{attribute 'TcRpcEnable' := '1'}
METHOD start
  VAR_INPUT
    position : LREAL;  (* New position setpoint *)
    maxVelocity : LREAL;  (* Maximum velocity *)
  END_VAR
                  THIS^.get.position := position;
THIS^.get.maxVelocity := maxVelocity;
THIS^.statuses.busyStatus( isBusy := TRUE );
THIS^.statuses.healthStatus( isGood := TRUE );

                
END_METHOD

{attribute 'TcRpcEnable' := '1'}
METHOD request : RequestResults
  VAR_INPUT
    position : LREAL;  (* New position setpoint *)
    maxVelocity : LREAL;  (* Maximum velocity *)
  END_VAR
                  IF THIS^.statuses.enabledStatus.enabled THEN
    THIS^.start(
        position := position,
        maxVelocity := maxVelocity);
    request := RequestResults.ACCEPTED;
ELSE
    request := RequestResults.REJECTED;
END_IF;

                
END_METHOD
END_FUNCTION_BLOCK

FUNCTION_BLOCK McMoveRelativeProcess EXTENDS BaseMcProcess
  VAR_INPUT
    {attribute 'OPC.UA.DA' := '1'}
    set : McMoveRelativeProcessArgs;  (* Arguments to be set, before writing do_request TRUE *)
  END_VAR
  VAR_OUTPUT
    {attribute 'OPC.UA.DA' := '1'}
    {attribute 'OPC.UA.DA.Access' := '1'}
    get : McMoveRelativeProcessArgs;  (* Arguments in use by the process, if do_request was accepted *)
  END_VAR

            IF do_request THEN
    do_request_result := request(
    distance := set.distance,
    maxVelocity := set.maxVelocity);
    do_request := FALSE;
END_IF;
SUPER^();

          

{attribute 'TcRpcEnable' := '1'}
METHOD start
  VAR_INPUT
    distance : LREAL;  (* Distance to move *)
    maxVelocity : LREAL;  (* Maximum velocity *)
  END_VAR
                  THIS^.get.distance := distance;
THIS^.get.maxVelocity := maxVelocity;
THIS^.statuses.busyStatus( isBusy := TRUE );
THIS^.statuses.healthStatus( isGood := TRUE );

                
END_METHOD

{attribute 'TcRpcEnable' := '1'}
METHOD request : RequestResults
  VAR_INPUT
    distance : LREAL;  (* Distance to move *)
    maxVelocity : LREAL;  (* Maximum velocity *)
  END_VAR
                  IF THIS^.statuses.enabledStatus.enabled THEN
    THIS^.start(
        distance := distance,
        maxVelocity := maxVelocity);
    request := RequestResults.ACCEPTED;
ELSE
    request := RequestResults.REJECTED;
END_IF;

                
END_METHOD
END_FUNCTION_BLOCK

FUNCTION_BLOCK McPowerProcess EXTENDS BaseMcProcess
  VAR_INPUT
    {attribute 'OPC.UA.DA' := '1'}
    set : McPowerProcessArgs;  (* Arguments to be set, before writing do_request TRUE *)
  END_VAR
  VAR_OUTPUT
    {attribute 'OPC.UA.DA' := '1'}
    {attribute 'OPC.UA.DA.Access' := '1'}
    get : McPowerProcessArgs;  (* Arguments in use by the process, if do_request was accepted *)
  END_VAR

            IF do_request THEN
    do_request_result := request( enable := set.enable );
    do_request := FALSE;
END_IF;
SUPER^();

          

{attribute 'TcRpcEnable' := '1'}
METHOD start
  VAR_INPUT
    enable : BOOL;  (* Enable the power or not *)
  END_VAR
                  THIS^.get.enable := enable;
THIS^.statuses.busyStatus( isBusy := TRUE );
THIS^.statuses.healthStatus( isGood := TRUE );

                
END_METHOD

{attribute 'TcRpcEnable' := '1'}
METHOD request : RequestResults
  VAR_INPUT
    enable : BOOL;  (* Enable the power or not *)
  END_VAR
                  IF THIS^.statuses.enabledStatus.enabled THEN
    THIS^.start( enable := enable );
    request := RequestResults.ACCEPTED;
ELSE
    request := RequestResults.REJECTED;
END_IF;

                
END_METHOD
END_FUNCTION_BLOCK

FUNCTION_BLOCK McSetPositionProcess EXTENDS BaseMcProcess
  VAR_INPUT
    {attribute 'OPC.UA.DA' := '1'}
    set : McSetPositionProcessArgs;  (* Arguments to be set, before writing do_request TRUE *)
  END_VAR
  VAR_OUTPUT
    {attribute 'OPC.UA.DA' := '1'}
    {attribute 'OPC.UA.DA.Access' := '1'}
    get : McSetPositionProcessArgs;  (* Arguments in use by the process, if do_request was accepted *)
  END_VAR

            IF do_request THEN
    do_request_result := request( value := set.value );
    do_request := FALSE;
END_IF;
SUPER^();

          

{attribute 'TcRpcEnable' := '1'}
METHOD start
  VAR_INPUT
    value : LREAL;  (* New position to be taken over by the encoder *)
  END_VAR
                  THIS^.get.value := value;
THIS^.statuses.busyStatus( isBusy := TRUE );
THIS^.statuses.healthStatus( isGood := TRUE );

                
END_METHOD

{attribute 'TcRpcEnable' := '1'}
METHOD request : RequestResults
  VAR_INPUT
    value : LREAL;  (* New position to be taken over by the encoder *)
  END_VAR
                  IF THIS^.statuses.enabledStatus.enabled THEN
    THIS^.start( value := value );
    request := RequestResults.ACCEPTED;
ELSE
    request := RequestResults.REJECTED;
END_IF;

                
END_METHOD
END_FUNCTION_BLOCK

FUNCTION_BLOCK McStopProcess EXTENDS BaseMcProcess
  VAR_INPUT
    {attribute 'OPC.UA.DA' := '1'}
    set : McStopProcessArgs;  (* Arguments to be set, before writing do_request TRUE *)
  END_VAR
  VAR_OUTPUT
    {attribute 'OPC.UA.DA' := '1'}
    {attribute 'OPC.UA.DA.Access' := '1'}
    get : McStopProcessArgs;  (* Arguments in use by the process, if do_request was accepted *)
  END_VAR

            IF do_request THEN
    do_request_result := request(
    deceleration := set.deceleration,
    jerk := set.jerk);
    do_request := FALSE;
END_IF;
SUPER^();

          

{attribute 'TcRpcEnable' := '1'}
METHOD start
  VAR_INPUT
    deceleration : LREAL;  (* Deceleration (use 0 for default). If non zero, then also jerk must be non zero! *)
    jerk : LREAL;  (* Jerk (use 0 for default). If non zero, then also deceleration must be non zero! *)
  END_VAR
                  THIS^.get.deceleration := deceleration;
THIS^.get.jerk := jerk;
THIS^.statuses.busyStatus( isBusy := TRUE );
THIS^.statuses.healthStatus( isGood := TRUE );

                
END_METHOD

{attribute 'TcRpcEnable' := '1'}
METHOD request : RequestResults
  VAR_INPUT
    deceleration : LREAL;  (* Deceleration (use 0 for default). If non zero, then also jerk must be non zero! *)
    jerk : LREAL;  (* Jerk (use 0 for default). If non zero, then also deceleration must be non zero! *)
  END_VAR
                  IF THIS^.statuses.enabledStatus.enabled THEN
    THIS^.start(
        deceleration := deceleration,
        jerk := jerk);
    request := RequestResults.ACCEPTED;
ELSE
    request := RequestResults.REJECTED;
END_IF;

                
END_METHOD
END_FUNCTION_BLOCK

FUNCTION_BLOCK McMoveVelocityProcess EXTENDS BaseMcProcess
  VAR_INPUT
    {attribute 'OPC.UA.DA' := '1'}
    set : McMoveVelocityProcessArgs;  (* Arguments to be set, before writing do_request TRUE *)
  END_VAR
  VAR_OUTPUT
    {attribute 'OPC.UA.DA' := '1'}
    {attribute 'OPC.UA.DA.Access' := '1'}
    get : McMoveVelocityProcessArgs;  (* Arguments in use by the process, if do_request was accepted *)
  END_VAR

            IF do_request THEN
    do_request_result := request( value := set.value );
    do_request := FALSE;
END_IF;
SUPER^();

          

{attribute 'TcRpcEnable' := '1'}
METHOD start
  VAR_INPUT
    value : LREAL;  (* New velocity *)
  END_VAR
                  THIS^.get.value := value;
THIS^.statuses.busyStatus( isBusy := TRUE );
THIS^.statuses.healthStatus( isGood := TRUE );

                
END_METHOD

{attribute 'TcRpcEnable' := '1'}
METHOD request : RequestResults
  VAR_INPUT
    value : LREAL;  (* New velocity *)
  END_VAR
                  IF THIS^.statuses.enabledStatus.enabled THEN
    THIS^.start( value := value );
    request := RequestResults.ACCEPTED;
ELSE
    request := RequestResults.REJECTED;
END_IF;

                
END_METHOD
END_FUNCTION_BLOCK

FUNCTION_BLOCK SetEnabledProcess EXTENDS BaseProcess
  VAR_INPUT
    {attribute 'OPC.UA.DA' := '1'}
    set : SetEnabledProcessArgs;  (* Arguments to be set, before writing do_request TRUE *)
  END_VAR
  VAR_OUTPUT
    {attribute 'OPC.UA.DA' := '1'}
    {attribute 'OPC.UA.DA.Access' := '1'}
    get : SetEnabledProcessArgs;  (* Arguments in use by the process, if do_request was accepted *)
  END_VAR

            IF do_request THEN
    do_request_result := request( enabled := set.enabled );
    do_request := FALSE;
END_IF;
SUPER^();

          

{attribute 'TcRpcEnable' := '1'}
METHOD start
  VAR_INPUT
    enabled : BOOL;  (* True to enable, false to disable *)
  END_VAR
                  THIS^.get.enabled := enabled;
THIS^.statuses.busyStatus( isBusy := TRUE );
THIS^.statuses.healthStatus( isGood := TRUE );

                
END_METHOD

{attribute 'TcRpcEnable' := '1'}
METHOD request : RequestResults
  VAR_INPUT
    enabled : BOOL;  (* True to enable, false to disable *)
  END_VAR
                  IF THIS^.statuses.enabledStatus.enabled THEN
    THIS^.start( enabled := enabled );
    request := RequestResults.ACCEPTED;
ELSE
    request := RequestResults.REJECTED;
END_IF;

                
END_METHOD
END_FUNCTION_BLOCK

FUNCTION_BLOCK McWriteParameter EXTENDS BaseMcProcess
  VAR_INPUT
    {attribute 'OPC.UA.DA' := '1'}
    set : McWriteParameterArgs;  (* Arguments to be set, before writing do_request TRUE *)
  END_VAR
  VAR_OUTPUT
    {attribute 'OPC.UA.DA' := '1'}
    {attribute 'OPC.UA.DA.Access' := '1'}
    get : McWriteParameterArgs;  (* Arguments in use by the process, if do_request was accepted *)
  END_VAR

            IF do_request THEN
    do_request_result := request(
    parameterNumber := set.parameterNumber,
    value := set.value);
    do_request := FALSE;
END_IF;
SUPER^();

          

{attribute 'TcRpcEnable' := '1'}
METHOD start
  VAR_INPUT
    parameterNumber : INT;  (* Number of the parameter *)
    value : LREAL;  (* Value to write *)
  END_VAR
                  THIS^.get.parameterNumber := parameterNumber;
THIS^.get.value := value;
THIS^.statuses.busyStatus( isBusy := TRUE );
THIS^.statuses.healthStatus( isGood := TRUE );

                
END_METHOD

{attribute 'TcRpcEnable' := '1'}
METHOD request : RequestResults
  VAR_INPUT
    parameterNumber : INT;  (* Number of the parameter *)
    value : LREAL;  (* Value to write *)
  END_VAR
                  IF THIS^.statuses.enabledStatus.enabled THEN
    THIS^.start(
        parameterNumber := parameterNumber,
        value := value);
    request := RequestResults.ACCEPTED;
ELSE
    request := RequestResults.REJECTED;
END_IF;

                
END_METHOD
END_FUNCTION_BLOCK

FUNCTION_BLOCK McReadParameter EXTENDS BaseMcProcess
  VAR_INPUT
    value : LREAL;  (* Value that was read *)
    {attribute 'OPC.UA.DA' := '1'}
    set : McReadParameterArgs;  (* Arguments to be set, before writing do_request TRUE *)
  END_VAR
  VAR_OUTPUT
    {attribute 'OPC.UA.DA' := '1'}
    {attribute 'OPC.UA.DA.Access' := '1'}
    get : McReadParameterArgs;  (* Arguments in use by the process, if do_request was accepted *)
  END_VAR

            IF do_request THEN
    do_request_result := request( parameterNumber := set.parameterNumber );
    do_request := FALSE;
END_IF;
SUPER^();

          

{attribute 'TcRpcEnable' := '1'}
METHOD start
  VAR_INPUT
    parameterNumber : INT;  (* Number of the parameter *)
  END_VAR
                  THIS^.get.parameterNumber := parameterNumber;
THIS^.statuses.busyStatus( isBusy := TRUE );
THIS^.statuses.healthStatus( isGood := TRUE );

                
END_METHOD

{attribute 'TcRpcEnable' := '1'}
METHOD request : RequestResults
  VAR_INPUT
    parameterNumber : INT;  (* Number of the parameter *)
  END_VAR
                  IF THIS^.statuses.enabledStatus.enabled THEN
    THIS^.start( parameterNumber := parameterNumber );
    request := RequestResults.ACCEPTED;
ELSE
    request := RequestResults.REJECTED;
END_IF;

                
END_METHOD
END_FUNCTION_BLOCK

FUNCTION_BLOCK McWriteBoolParameter EXTENDS BaseMcProcess
  VAR_INPUT
    {attribute 'OPC.UA.DA' := '1'}
    set : McWriteBoolParameterArgs;  (* Arguments to be set, before writing do_request TRUE *)
  END_VAR
  VAR_OUTPUT
    {attribute 'OPC.UA.DA' := '1'}
    {attribute 'OPC.UA.DA.Access' := '1'}
    get : McWriteBoolParameterArgs;  (* Arguments in use by the process, if do_request was accepted *)
  END_VAR

            IF do_request THEN
    do_request_result := request(
    parameterNumber := set.parameterNumber,
    value := set.value);
    do_request := FALSE;
END_IF;
SUPER^();

          

{attribute 'TcRpcEnable' := '1'}
METHOD start
  VAR_INPUT
    parameterNumber : INT;  (* Number of the parameter *)
    value : BOOL;  (* Value to write *)
  END_VAR
                  THIS^.get.parameterNumber := parameterNumber;
THIS^.get.value := value;
THIS^.statuses.busyStatus( isBusy := TRUE );
THIS^.statuses.healthStatus( isGood := TRUE );

                
END_METHOD

{attribute 'TcRpcEnable' := '1'}
METHOD request : RequestResults
  VAR_INPUT
    parameterNumber : INT;  (* Number of the parameter *)
    value : BOOL;  (* Value to write *)
  END_VAR
                  IF THIS^.statuses.enabledStatus.enabled THEN
    THIS^.start(
        parameterNumber := parameterNumber,
        value := value);
    request := RequestResults.ACCEPTED;
ELSE
    request := RequestResults.REJECTED;
END_IF;

                
END_METHOD
END_FUNCTION_BLOCK

FUNCTION_BLOCK McReadBoolParameter EXTENDS BaseMcProcess
  VAR_INPUT
    value : BOOL;  (* Value that was read *)
    {attribute 'OPC.UA.DA' := '1'}
    set : McReadBoolParameterArgs;  (* Arguments to be set, before writing do_request TRUE *)
  END_VAR
  VAR_OUTPUT
    {attribute 'OPC.UA.DA' := '1'}
    {attribute 'OPC.UA.DA.Access' := '1'}
    get : McReadBoolParameterArgs;  (* Arguments in use by the process, if do_request was accepted *)
  END_VAR

            IF do_request THEN
    do_request_result := request( parameterNumber := set.parameterNumber );
    do_request := FALSE;
END_IF;
SUPER^();

          

{attribute 'TcRpcEnable' := '1'}
METHOD start
  VAR_INPUT
    parameterNumber : INT;  (* Number of the parameter *)
  END_VAR
                  THIS^.get.parameterNumber := parameterNumber;
THIS^.statuses.busyStatus( isBusy := TRUE );
THIS^.statuses.healthStatus( isGood := TRUE );

                
END_METHOD

{attribute 'TcRpcEnable' := '1'}
METHOD request : RequestResults
  VAR_INPUT
    parameterNumber : INT;  (* Number of the parameter *)
  END_VAR
                  IF THIS^.statuses.enabledStatus.enabled THEN
    THIS^.start( parameterNumber := parameterNumber );
    request := RequestResults.ACCEPTED;
ELSE
    request := RequestResults.REJECTED;
END_IF;

                
END_METHOD
END_FUNCTION_BLOCK

FUNCTION_BLOCK SDOReadProcess EXTENDS BaseProcess
  VAR_INPUT
    value1Byte : USINT;  (* Value that has been read, if noOfBytes is 1 *)
    value2Bytes : UINT;  (* Value that has been read, if noOfBytes is 2 *)
    value4Bytes : UDINT;  (* Value that has been read, if noOfBytes is 4 *)
    errorId : UDINT;  (* Error ID according to Beckhoff *)
    {attribute 'OPC.UA.DA' := '1'}
    set : SDOReadProcessArgs;  (* Arguments to be set, before writing do_request TRUE *)
  END_VAR
  VAR_OUTPUT
    {attribute 'OPC.UA.DA' := '1'}
    {attribute 'OPC.UA.DA.Access' := '1'}
    get : SDOReadProcessArgs;  (* Arguments in use by the process, if do_request was accepted *)
  END_VAR

            IF do_request THEN
    do_request_result := request(
    index := set.index,
    subindex := set.subindex,
    noOfBytes := set.noOfBytes);
    do_request := FALSE;
END_IF;
SUPER^();

          

{attribute 'TcRpcEnable' := '1'}
METHOD start
  VAR_INPUT
    index : UINT;  (* SDO Index *)
    subindex : USINT;  (* SDO SubIndex *)
    noOfBytes : UDINT;  (* Number of bytes to be read *)
  END_VAR
                  THIS^.get.index := index;
THIS^.get.subindex := subindex;
THIS^.get.noOfBytes := noOfBytes;
THIS^.statuses.busyStatus( isBusy := TRUE );
THIS^.statuses.healthStatus( isGood := TRUE );

                
END_METHOD

{attribute 'TcRpcEnable' := '1'}
METHOD request : RequestResults
  VAR_INPUT
    index : UINT;  (* SDO Index *)
    subindex : USINT;  (* SDO SubIndex *)
    noOfBytes : UDINT;  (* Number of bytes to be read *)
  END_VAR
                  IF THIS^.statuses.enabledStatus.enabled THEN
    THIS^.start(
        index := index,
        subindex := subindex,
        noOfBytes := noOfBytes);
    request := RequestResults.ACCEPTED;
ELSE
    request := RequestResults.REJECTED;
END_IF;

                
END_METHOD
END_FUNCTION_BLOCK

FUNCTION_BLOCK SDOWriteProcess EXTENDS BaseProcess
  VAR_INPUT
    errorId : UDINT;  (* Error ID according to Beckhoff *)
    {attribute 'OPC.UA.DA' := '1'}
    set : SDOWriteProcessArgs;  (* Arguments to be set, before writing do_request TRUE *)
  END_VAR
  VAR_OUTPUT
    {attribute 'OPC.UA.DA' := '1'}
    {attribute 'OPC.UA.DA.Access' := '1'}
    get : SDOWriteProcessArgs;  (* Arguments in use by the process, if do_request was accepted *)
  END_VAR

            IF do_request THEN
    do_request_result := request(
    index := set.index,
    subindex := set.subindex,
    noOfBytes := set.noOfBytes,
    value1Byte := set.value1Byte,
    value2Bytes := set.value2Bytes,
    value4Bytes := set.value4Bytes);
    do_request := FALSE;
END_IF;
SUPER^();

          

{attribute 'TcRpcEnable' := '1'}
METHOD start
  VAR_INPUT
    index : UINT;  (* SDO Index *)
    subindex : USINT;  (* SDO SubIndex *)
    noOfBytes : UDINT;  (* Number of bytes to be written *)
    value1Byte : USINT;  (* Value to be written if noOfBytes is 1 *)
    value2Bytes : UINT;  (* Value to be written if noOfBytes is 2 *)
    value4Bytes : UDINT;  (* Value to be written if noOfBytes is 4 *)
  END_VAR
                  THIS^.get.index := index;
THIS^.get.subindex := subindex;
THIS^.get.noOfBytes := noOfBytes;
THIS^.get.value1Byte := value1Byte;
THIS^.get.value2Bytes := value2Bytes;
THIS^.get.value4Bytes := value4Bytes;
THIS^.statuses.busyStatus( isBusy := TRUE );
THIS^.statuses.healthStatus( isGood := TRUE );

                
END_METHOD

{attribute 'TcRpcEnable' := '1'}
METHOD request : RequestResults
  VAR_INPUT
    index : UINT;  (* SDO Index *)
    subindex : USINT;  (* SDO SubIndex *)
    noOfBytes : UDINT;  (* Number of bytes to be written *)
    value1Byte : USINT;  (* Value to be written if noOfBytes is 1 *)
    value2Bytes : UINT;  (* Value to be written if noOfBytes is 2 *)
    value4Bytes : UDINT;  (* Value to be written if noOfBytes is 4 *)
  END_VAR
                  IF THIS^.statuses.enabledStatus.enabled THEN
    THIS^.start(
        index := index,
        subindex := subindex,
        noOfBytes := noOfBytes,
        value1Byte := value1Byte,
        value2Bytes := value2Bytes,
        value4Bytes := value4Bytes);
    request := RequestResults.ACCEPTED;
ELSE
    request := RequestResults.REJECTED;
END_IF;

                
END_METHOD
END_FUNCTION_BLOCK

FUNCTION_BLOCK SoEReadProcess EXTENDS BaseProcess
  VAR_INPUT
    value1Byte : USINT;  (* Value that has been read, if noOfBytes is 1 *)
    value2Bytes : UINT;  (* Value that has been read, if noOfBytes is 2 *)
    value4Bytes : UDINT;  (* Value that has been read, if noOfBytes is 4 *)
    adsErrorId : UINT;  (* ADS error ID *)
    sercosErrorId : UINT;  (* Sercos error ID *)
    {attribute 'OPC.UA.DA' := '1'}
    set : SoEReadProcessArgs;  (* Arguments to be set, before writing do_request TRUE *)
  END_VAR
  VAR_OUTPUT
    {attribute 'OPC.UA.DA' := '1'}
    {attribute 'OPC.UA.DA.Access' := '1'}
    get : SoEReadProcessArgs;  (* Arguments in use by the process, if do_request was accepted *)
  END_VAR

            IF do_request THEN
    do_request_result := request(
    index := set.index,
    noOfBytes := set.noOfBytes);
    do_request := FALSE;
END_IF;
SUPER^();

          

{attribute 'TcRpcEnable' := '1'}
METHOD start
  VAR_INPUT
    index : UINT;  (* SDO Index *)
    noOfBytes : UDINT;  (* Number of bytes to be read *)
  END_VAR
                  THIS^.get.index := index;
THIS^.get.noOfBytes := noOfBytes;
THIS^.statuses.busyStatus( isBusy := TRUE );
THIS^.statuses.healthStatus( isGood := TRUE );

                
END_METHOD

{attribute 'TcRpcEnable' := '1'}
METHOD request : RequestResults
  VAR_INPUT
    index : UINT;  (* SDO Index *)
    noOfBytes : UDINT;  (* Number of bytes to be read *)
  END_VAR
                  IF THIS^.statuses.enabledStatus.enabled THEN
    THIS^.start(
        index := index,
        noOfBytes := noOfBytes);
    request := RequestResults.ACCEPTED;
ELSE
    request := RequestResults.REJECTED;
END_IF;

                
END_METHOD
END_FUNCTION_BLOCK

FUNCTION_BLOCK SoEWriteProcess EXTENDS BaseProcess
  VAR_INPUT
    adsErrorId : UINT;  (* ADS error ID *)
    sercosErrorId : UINT;  (* Sercos error ID *)
    {attribute 'OPC.UA.DA' := '1'}
    set : SoEWriteProcessArgs;  (* Arguments to be set, before writing do_request TRUE *)
  END_VAR
  VAR_OUTPUT
    {attribute 'OPC.UA.DA' := '1'}
    {attribute 'OPC.UA.DA.Access' := '1'}
    get : SoEWriteProcessArgs;  (* Arguments in use by the process, if do_request was accepted *)
  END_VAR

            IF do_request THEN
    do_request_result := request(
    index := set.index,
    noOfBytes := set.noOfBytes,
    value1Byte := set.value1Byte,
    value2Bytes := set.value2Bytes,
    value4Bytes := set.value4Bytes);
    do_request := FALSE;
END_IF;
SUPER^();

          

{attribute 'TcRpcEnable' := '1'}
METHOD start
  VAR_INPUT
    index : UINT;  (* SDO Index *)
    noOfBytes : UDINT;  (* Number of bytes to be written *)
    value1Byte : USINT;  (* Value to be written if noOfBytes is 1 *)
    value2Bytes : UINT;  (* Value to be written if noOfBytes is 2 *)
    value4Bytes : UDINT;  (* Value to be written if noOfBytes is 4 *)
  END_VAR
                  THIS^.get.index := index;
THIS^.get.noOfBytes := noOfBytes;
THIS^.get.value1Byte := value1Byte;
THIS^.get.value2Bytes := value2Bytes;
THIS^.get.value4Bytes := value4Bytes;
THIS^.statuses.busyStatus( isBusy := TRUE );
THIS^.statuses.healthStatus( isGood := TRUE );

                
END_METHOD

{attribute 'TcRpcEnable' := '1'}
METHOD request : RequestResults
  VAR_INPUT
    index : UINT;  (* SDO Index *)
    noOfBytes : UDINT;  (* Number of bytes to be written *)
    value1Byte : USINT;  (* Value to be written if noOfBytes is 1 *)
    value2Bytes : UINT;  (* Value to be written if noOfBytes is 2 *)
    value4Bytes : UDINT;  (* Value to be written if noOfBytes is 4 *)
  END_VAR
                  IF THIS^.statuses.enabledStatus.enabled THEN
    THIS^.start(
        index := index,
        noOfBytes := noOfBytes,
        value1Byte := value1Byte,
        value2Bytes := value2Bytes,
        value4Bytes := value4Bytes);
    request := RequestResults.ACCEPTED;
ELSE
    request := RequestResults.REJECTED;
END_IF;

                
END_METHOD
END_FUNCTION_BLOCK

FUNCTION_BLOCK SoEResetProcess EXTENDS BaseProcess
  VAR_INPUT
    adsErrorId : UINT;  (* ADS error ID *)
    sercosErrorId : UINT;  (* Sercos error ID *)
  END_VAR

            IF do_request THEN
    do_request_result := request();
    do_request := FALSE;
END_IF;
SUPER^();

          

{attribute 'TcRpcEnable' := '1'}
METHOD start
                  THIS^.statuses.busyStatus( isBusy := TRUE );
THIS^.statuses.healthStatus( isGood := TRUE );

                
END_METHOD

{attribute 'TcRpcEnable' := '1'}
METHOD request : RequestResults
                  IF THIS^.statuses.enabledStatus.enabled THEN
    THIS^.start();
    request := RequestResults.ACCEPTED;
ELSE
    request := RequestResults.REJECTED;
END_IF;

                
END_METHOD
END_FUNCTION_BLOCK

FUNCTION_BLOCK SetBrakeProcess EXTENDS BaseProcess
  VAR_INPUT
    {attribute 'OPC.UA.DA' := '1'}
    set : SetBrakeProcessArgs;  (* Arguments to be set, before writing do_request TRUE *)
  END_VAR
  VAR_OUTPUT
    {attribute 'OPC.UA.DA' := '1'}
    {attribute 'OPC.UA.DA.Access' := '1'}
    get : SetBrakeProcessArgs;  (* Arguments in use by the process, if do_request was accepted *)
  END_VAR

            IF do_request THEN
    do_request_result := request( newState := set.newState );
    do_request := FALSE;
END_IF;
SUPER^();

          

{attribute 'TcRpcEnable' := '1'}
METHOD start
  VAR_INPUT
    newState : DriveBrakeStates;  (* Requested brake state *)
  END_VAR
                  THIS^.get.newState := newState;
THIS^.statuses.busyStatus( isBusy := TRUE );
THIS^.statuses.healthStatus( isGood := TRUE );

                
END_METHOD

{attribute 'TcRpcEnable' := '1'}
METHOD request : RequestResults
  VAR_INPUT
    newState : DriveBrakeStates;  (* Requested brake state *)
  END_VAR
                  IF THIS^.statuses.enabledStatus.enabled THEN
    THIS^.start( newState := newState );
    request := RequestResults.ACCEPTED;
ELSE
    request := RequestResults.REJECTED;
END_IF;

                
END_METHOD
END_FUNCTION_BLOCK

FUNCTION_BLOCK ChangeOperatingStateProcess EXTENDS BaseProcess
  VAR_INPUT
    {attribute 'OPC.UA.DA' := '1'}
    set : ChangeOperatingStateProcessArgs;  (* Arguments to be set, before writing do_request TRUE *)
  END_VAR
  VAR_OUTPUT
    {attribute 'OPC.UA.DA' := '1'}
    {attribute 'OPC.UA.DA.Access' := '1'}
    get : ChangeOperatingStateProcessArgs;  (* Arguments in use by the process, if do_request was accepted *)
  END_VAR

            IF do_request THEN
    do_request_result := request( state := set.state );
    do_request := FALSE;
END_IF;
SUPER^();

          

{attribute 'TcRpcEnable' := '1'}
METHOD start
  VAR_INPUT
    state : OperatingStates;  (* New operating state (e.g. AUTO, MANUAL) *)
  END_VAR
                  THIS^.get.state := state;
THIS^.statuses.busyStatus( isBusy := TRUE );
THIS^.statuses.healthStatus( isGood := TRUE );

                
END_METHOD

{attribute 'TcRpcEnable' := '1'}
METHOD request : RequestResults
  VAR_INPUT
    state : OperatingStates;  (* New operating state (e.g. AUTO, MANUAL) *)
  END_VAR
                  IF THIS^.statuses.enabledStatus.enabled THEN
    THIS^.start( state := state );
    request := RequestResults.ACCEPTED;
ELSE
    request := RequestResults.REJECTED;
END_IF;

                
END_METHOD
END_FUNCTION_BLOCK

FUNCTION_BLOCK ChangeOperatorStateProcess EXTENDS BaseProcess
  VAR_INPUT
    {attribute 'OPC.UA.DA' := '1'}
    set : ChangeOperatorStateProcessArgs;  (* Arguments to be set, before writing do_request TRUE *)
  END_VAR
  VAR_OUTPUT
    {attribute 'OPC.UA.DA' := '1'}
    {attribute 'OPC.UA.DA.Access' := '1'}
    get : ChangeOperatorStateProcessArgs;  (* Arguments in use by the process, if do_request was accepted *)
  END_VAR

            IF do_request THEN
    do_request_result := request(
    state := set.state,
    password := set.password);
    do_request := FALSE;
END_IF;
SUPER^();

          

{attribute 'TcRpcEnable' := '1'}
METHOD start
  VAR_INPUT
    state : OperatorStates;  (* New operator state (e.g. OBSERVER, TECH, ...) *)
    password : STRING;  (* Password (only sometimes required, e.g. to go from OBSERVER to TECH) *)
  END_VAR
                  THIS^.get.state := state;
THIS^.get.password := password;
THIS^.statuses.busyStatus( isBusy := TRUE );
THIS^.statuses.healthStatus( isGood := TRUE );

                
END_METHOD

{attribute 'TcRpcEnable' := '1'}
METHOD request : RequestResults
  VAR_INPUT
    state : OperatorStates;  (* New operator state (e.g. OBSERVER, TECH, ...) *)
    password : STRING;  (* Password (only sometimes required, e.g. to go from OBSERVER to TECH) *)
  END_VAR
                  IF THIS^.statuses.enabledStatus.enabled THEN
    THIS^.start(
        state := state,
        password := password);
    request := RequestResults.ACCEPTED;
ELSE
    request := RequestResults.REJECTED;
END_IF;

                
END_METHOD
END_FUNCTION_BLOCK

FUNCTION_BLOCK ReadXmlProcess EXTENDS BaseXmlDataSrvProcess
  VAR_INPUT
    {attribute 'OPC.UA.DA' := '1'}
    set : ReadXmlProcessArgs;  (* Arguments to be set, before writing do_request TRUE *)
  END_VAR
  VAR_OUTPUT
    {attribute 'OPC.UA.DA' := '1'}
    {attribute 'OPC.UA.DA.Access' := '1'}
    get : ReadXmlProcessArgs;  (* Arguments in use by the process, if do_request was accepted *)
  END_VAR

            IF do_request THEN
    do_request_result := request( filePath := set.filePath );
    do_request := FALSE;
END_IF;
SUPER^();

          

{attribute 'TcRpcEnable' := '1'}
METHOD start
  VAR_INPUT
    filePath : STRING;  (* Full path of the filename to read *)
  END_VAR
                  THIS^.get.filePath := filePath;
THIS^.statuses.busyStatus( isBusy := TRUE );
THIS^.statuses.healthStatus( isGood := TRUE );

                
END_METHOD

{attribute 'TcRpcEnable' := '1'}
METHOD request : RequestResults
  VAR_INPUT
    filePath : STRING;  (* Full path of the filename to read *)
  END_VAR
                  IF THIS^.statuses.enabledStatus.enabled THEN
    THIS^.start( filePath := filePath );
    request := RequestResults.ACCEPTED;
ELSE
    request := RequestResults.REJECTED;
END_IF;

                
END_METHOD
END_FUNCTION_BLOCK

FUNCTION_BLOCK WriteXmlProcess EXTENDS BaseXmlDataSrvProcess
  VAR_INPUT
    {attribute 'OPC.UA.DA' := '1'}
    set : WriteXmlProcessArgs;  (* Arguments to be set, before writing do_request TRUE *)
  END_VAR
  VAR_OUTPUT
    {attribute 'OPC.UA.DA' := '1'}
    {attribute 'OPC.UA.DA.Access' := '1'}
    get : WriteXmlProcessArgs;  (* Arguments in use by the process, if do_request was accepted *)
  END_VAR

            IF do_request THEN
    do_request_result := request( filePath := set.filePath );
    do_request := FALSE;
END_IF;
SUPER^();

          

{attribute 'TcRpcEnable' := '1'}
METHOD start
  VAR_INPUT
    filePath : STRING;  (* Full path of the filename to write *)
  END_VAR
                  THIS^.get.filePath := filePath;
THIS^.statuses.busyStatus( isBusy := TRUE );
THIS^.statuses.healthStatus( isGood := TRUE );

                
END_METHOD

{attribute 'TcRpcEnable' := '1'}
METHOD request : RequestResults
  VAR_INPUT
    filePath : STRING;  (* Full path of the filename to write *)
  END_VAR
                  IF THIS^.statuses.enabledStatus.enabled THEN
    THIS^.start( filePath := filePath );
    request := RequestResults.ACCEPTED;
ELSE
    request := RequestResults.REJECTED;
END_IF;

                
END_METHOD
END_FUNCTION_BLOCK

FUNCTION_BLOCK ActivateProcess EXTENDS BaseProcess
  VAR
    {attribute 'OPC.UA.DA' := '0'}
    testVar : BOOL;  (* At least 1 variable needed because subclass members of an empty class are not exposed by OPC UA (TwinCAT bug!) *)
  END_VAR

            IF do_request THEN
    do_request_result := request();
    do_request := FALSE;
END_IF;
SUPER^();

          

{attribute 'TcRpcEnable' := '1'}
METHOD start
                  THIS^.statuses.busyStatus( isBusy := TRUE );
THIS^.statuses.healthStatus( isGood := TRUE );

                
END_METHOD

{attribute 'TcRpcEnable' := '1'}
METHOD request : RequestResults
                  IF THIS^.statuses.enabledStatus.enabled THEN
    THIS^.start();
    request := RequestResults.ACCEPTED;
ELSE
    request := RequestResults.REJECTED;
END_IF;

                
END_METHOD
END_FUNCTION_BLOCK

FUNCTION_BLOCK ModbusRTUBusReadCoilProcess EXTENDS BaseProcess
  VAR_INPUT
    value : BOOL;  (* Value of the coil *)
    errorId : INT;  (* Error Id. Modbus error code *)
    {attribute 'OPC.UA.DA' := '1'}
    set : ModbusRTUBusReadCoilProcessArgs;  (* Arguments to be set, before writing do_request TRUE *)
  END_VAR
  VAR_OUTPUT
    {attribute 'OPC.UA.DA' := '1'}
    {attribute 'OPC.UA.DA.Access' := '1'}
    get : ModbusRTUBusReadCoilProcessArgs;  (* Arguments in use by the process, if do_request was accepted *)
  END_VAR

            IF do_request THEN
    do_request_result := request(
    unitID := set.unitID,
    address := set.address);
    do_request := FALSE;
END_IF;
SUPER^();

          

{attribute 'TcRpcEnable' := '1'}
METHOD start
  VAR_INPUT
    unitID : USINT;  (* Modbus station address (1..247) *)
    address : UINT;  (* Modbus data address *)
  END_VAR
                  THIS^.get.unitID := unitID;
THIS^.get.address := address;
THIS^.statuses.busyStatus( isBusy := TRUE );
THIS^.statuses.healthStatus( isGood := TRUE );

                
END_METHOD

{attribute 'TcRpcEnable' := '1'}
METHOD request : RequestResults
  VAR_INPUT
    unitID : USINT;  (* Modbus station address (1..247) *)
    address : UINT;  (* Modbus data address *)
  END_VAR
                  IF THIS^.statuses.enabledStatus.enabled THEN
    THIS^.start(
        unitID := unitID,
        address := address);
    request := RequestResults.ACCEPTED;
ELSE
    request := RequestResults.REJECTED;
END_IF;

                
END_METHOD
END_FUNCTION_BLOCK

FUNCTION_BLOCK ModbusRTUBusWriteCoilProcess EXTENDS BaseProcess
  VAR_INPUT
    errorId : INT;  (* Error Id. Modbus error code *)
    {attribute 'OPC.UA.DA' := '1'}
    set : ModbusRTUBusWriteCoilProcessArgs;  (* Arguments to be set, before writing do_request TRUE *)
  END_VAR
  VAR_OUTPUT
    {attribute 'OPC.UA.DA' := '1'}
    {attribute 'OPC.UA.DA.Access' := '1'}
    get : ModbusRTUBusWriteCoilProcessArgs;  (* Arguments in use by the process, if do_request was accepted *)
  END_VAR

            IF do_request THEN
    do_request_result := request(
    unitID := set.unitID,
    address := set.address,
    value := set.value);
    do_request := FALSE;
END_IF;
SUPER^();

          

{attribute 'TcRpcEnable' := '1'}
METHOD start
  VAR_INPUT
    unitID : USINT;  (* Modbus station address (1..247) *)
    address : UINT;  (* Modbus data address *)
    value : BOOL;  (* Value to write on the coil *)
  END_VAR
                  THIS^.get.unitID := unitID;
THIS^.get.address := address;
THIS^.get.value := value;
THIS^.statuses.busyStatus( isBusy := TRUE );
THIS^.statuses.healthStatus( isGood := TRUE );

                
END_METHOD

{attribute 'TcRpcEnable' := '1'}
METHOD request : RequestResults
  VAR_INPUT
    unitID : USINT;  (* Modbus station address (1..247) *)
    address : UINT;  (* Modbus data address *)
    value : BOOL;  (* Value to write on the coil *)
  END_VAR
                  IF THIS^.statuses.enabledStatus.enabled THEN
    THIS^.start(
        unitID := unitID,
        address := address,
        value := value);
    request := RequestResults.ACCEPTED;
ELSE
    request := RequestResults.REJECTED;
END_IF;

                
END_METHOD
END_FUNCTION_BLOCK

FUNCTION_BLOCK ModbusRTUBusReadRegisterProcess EXTENDS BaseProcess
  VAR_INPUT
    value : INT;  (* Value of the register *)
    errorId : INT;  (* Error Id. Modbus error code *)
    {attribute 'OPC.UA.DA' := '1'}
    set : ModbusRTUBusReadRegisterProcessArgs;  (* Arguments to be set, before writing do_request TRUE *)
  END_VAR
  VAR_OUTPUT
    {attribute 'OPC.UA.DA' := '1'}
    {attribute 'OPC.UA.DA.Access' := '1'}
    get : ModbusRTUBusReadRegisterProcessArgs;  (* Arguments in use by the process, if do_request was accepted *)
  END_VAR

            IF do_request THEN
    do_request_result := request(
    unitID := set.unitID,
    address := set.address);
    do_request := FALSE;
END_IF;
SUPER^();

          

{attribute 'TcRpcEnable' := '1'}
METHOD start
  VAR_INPUT
    unitID : USINT;  (* Modbus station address (1..247) *)
    address : UINT;  (* Modbus data address *)
  END_VAR
                  THIS^.get.unitID := unitID;
THIS^.get.address := address;
THIS^.statuses.busyStatus( isBusy := TRUE );
THIS^.statuses.healthStatus( isGood := TRUE );

                
END_METHOD

{attribute 'TcRpcEnable' := '1'}
METHOD request : RequestResults
  VAR_INPUT
    unitID : USINT;  (* Modbus station address (1..247) *)
    address : UINT;  (* Modbus data address *)
  END_VAR
                  IF THIS^.statuses.enabledStatus.enabled THEN
    THIS^.start(
        unitID := unitID,
        address := address);
    request := RequestResults.ACCEPTED;
ELSE
    request := RequestResults.REJECTED;
END_IF;

                
END_METHOD
END_FUNCTION_BLOCK

FUNCTION_BLOCK ModbusRTUBusWriteRegisterProcess EXTENDS BaseProcess
  VAR_INPUT
    errorId : INT;  (* Error Id. Modbus error code *)
    {attribute 'OPC.UA.DA' := '1'}
    set : ModbusRTUBusWriteRegisterProcessArgs;  (* Arguments to be set, before writing do_request TRUE *)
  END_VAR
  VAR_OUTPUT
    {attribute 'OPC.UA.DA' := '1'}
    {attribute 'OPC.UA.DA.Access' := '1'}
    get : ModbusRTUBusWriteRegisterProcessArgs;  (* Arguments in use by the process, if do_request was accepted *)
  END_VAR

            IF do_request THEN
    do_request_result := request(
    unitID := set.unitID,
    address := set.address,
    value := set.value);
    do_request := FALSE;
END_IF;
SUPER^();

          

{attribute 'TcRpcEnable' := '1'}
METHOD start
  VAR_INPUT
    unitID : USINT;  (* Modbus station address (1..247) *)
    address : UINT;  (* Modbus data address *)
    value : INT;  (* Value to write on the register *)
  END_VAR
                  THIS^.get.unitID := unitID;
THIS^.get.address := address;
THIS^.get.value := value;
THIS^.statuses.busyStatus( isBusy := TRUE );
THIS^.statuses.healthStatus( isGood := TRUE );

                
END_METHOD

{attribute 'TcRpcEnable' := '1'}
METHOD request : RequestResults
  VAR_INPUT
    unitID : USINT;  (* Modbus station address (1..247) *)
    address : UINT;  (* Modbus data address *)
    value : INT;  (* Value to write on the register *)
  END_VAR
                  IF THIS^.statuses.enabledStatus.enabled THEN
    THIS^.start(
        unitID := unitID,
        address := address,
        value := value);
    request := RequestResults.ACCEPTED;
ELSE
    request := RequestResults.REJECTED;
END_IF;

                
END_METHOD
END_FUNCTION_BLOCK
